FUNCTION_BLOCK FB_HwRefDiluter
VAR_INPUT
	bIsInit 		: BOOL;
	bBusy			: BOOL;
	eValveType 		: E_DilValveType;
	nActValvePos	: SINT;
	nActPlungerPos	: UINT;	
END_VAR
VAR_OUTPUT
	nChannel		: USINT;
END_VAR
VAR
END_VAR
VAR_STAT
	nHighestChannel : USINT;
END_VAR

METHOD FB_init : BOOL
VAR_INPUT
	bInitRetains : BOOL; // if TRUE, the retain variables are initialized (warm start / cold start)
	bInCopyCode : BOOL;  // if TRUE, the instance afterwards gets moved into the copy code (online change)
END_VAR
nHighestChannel := nHighestChannel + 1;
nChannel := nHighestChannel;
END_METHOD

END_FUNCTION_BLOCK

(* stored: Version 1.1.0.1, ProductVersion 3.1.4022.10
   POU FB_HwRefDiluter: Id {727b2819-518c-4c5e-9c6b-f756216b1c19}, SpecialFunc None
   Method FB_init: Id {995e1476-433c-46e6-a922-2e154939e04c} *)
